TYPE ST_P_WAIT :
STRUCT
	WaitTime:		INT;
	ExecuteOnFail:	BOOL;
END_STRUCT
END_TYPE

(* stored: Version 1.1.0.1, ProductVersion 3.1.4024.10
   DUT ST_P_WAIT: Id {50df8764-8344-49d7-aa20-03bb064a4a9b} *)
